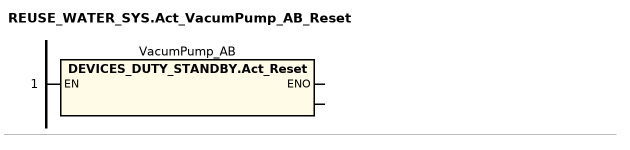
[picture p24: REUSE_WATER_SYS.Act_VacumPump_AB_Reset (LD)]
_LD_ (* Ladder Diagram *)
NETWORK 1
	*
		EN --- VacumPump_AB:DEVICES_DUTY_STANDBY.Act_Reset()
_END_LD_
(* the same logic as Structured Text *)
(* Network 1 *)
VacumPump_AB();
END_ACTION
ACTION Act_VacumPump_AB_Start:
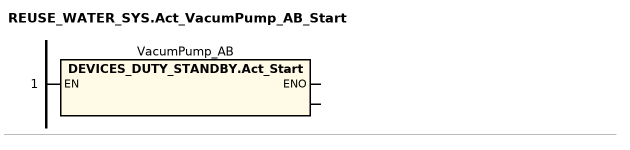
_LD_ (* Ladder Diagram *)
NETWORK 1
	*
		EN --- VacumPump_AB:DEVICES_DUTY_STANDBY.Act_Start()
_END_LD_
(* the same logic as Structured Text *)
(* Network 1 *)
VacumPump_AB();
END_ACTION
ACTION Act_VacumPump_AB_Stop:
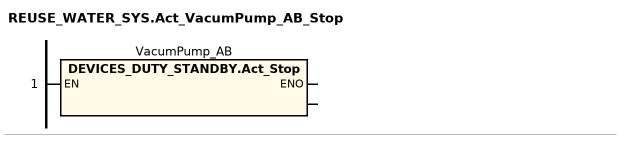
_LD_ (* Ladder Diagram *)
NETWORK 1
	*
		EN --- VacumPump_AB:DEVICES_DUTY_STANDBY.Act_Stop()
_END_LD_
(* the same logic as Structured Text *)
(* Network 1 *)
VacumPump_AB();
END_ACTION
ACTION Control:
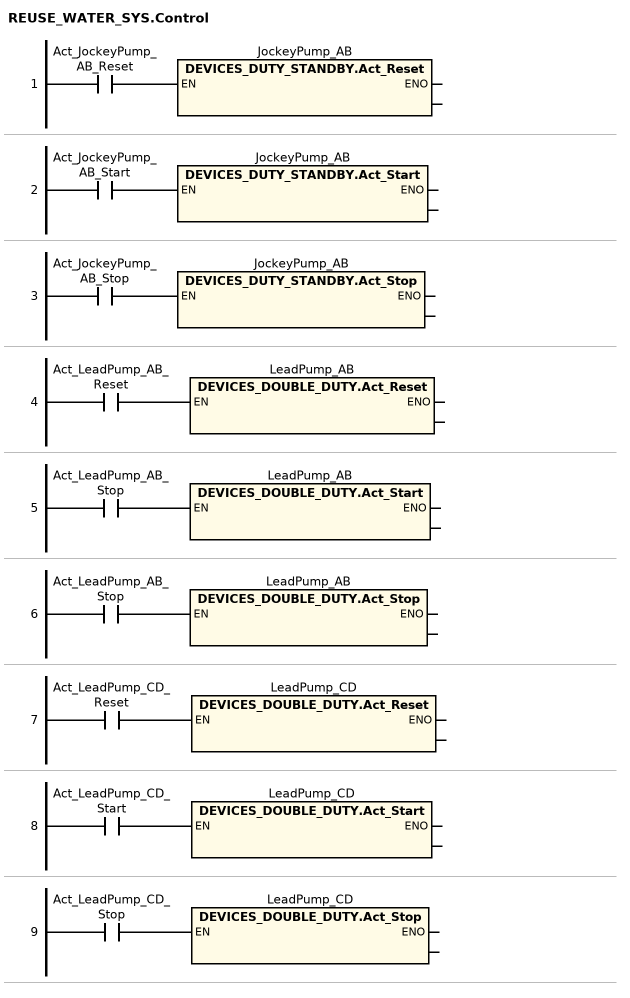
_LD_ (* Ladder Diagram *)
NETWORK 1
	[Act_JockeyPump_AB_Reset]
		EN --- JockeyPump_AB:DEVICES_DUTY_STANDBY.Act_Reset()
NETWORK 2
	[Act_JockeyPump_AB_Start]
		EN --- JockeyPump_AB:DEVICES_DUTY_STANDBY.Act_Start()
NETWORK 3
	[Act_JockeyPump_AB_Stop]
		EN --- JockeyPump_AB:DEVICES_DUTY_STANDBY.Act_Stop()
NETWORK 4
	[Act_LeadPump_AB_Reset]
		EN --- LeadPump_AB:DEVICES_DOUBLE_DUTY.Act_Reset()
NETWORK 5
	[Act_LeadPump_AB_Stop]
		EN --- LeadPump_AB:DEVICES_DOUBLE_DUTY.Act_Start()
NETWORK 6
	[Act_LeadPump_AB_Stop]
		EN --- LeadPump_AB:DEVICES_DOUBLE_DUTY.Act_Stop()
NETWORK 7
	[Act_LeadPump_CD_Reset]
		EN --- LeadPump_CD:DEVICES_DOUBLE_DUTY.Act_Reset()
NETWORK 8
	[Act_LeadPump_CD_Start]
		EN --- LeadPump_CD:DEVICES_DOUBLE_DUTY.Act_Start()
NETWORK 9
	[Act_LeadPump_CD_Stop]
		EN --- LeadPump_CD:DEVICES_DOUBLE_DUTY.Act_Stop()
_END_LD_
(* the same logic as Structured Text *)
(* Network 1 *)
IF Act_JockeyPump_AB_Reset THEN
	JockeyPump_AB();
END_IF;
(* Network 2 *)
IF Act_JockeyPump_AB_Start THEN
	JockeyPump_AB();
END_IF;
(* Network 3 *)
IF Act_JockeyPump_AB_Stop THEN
	JockeyPump_AB();
END_IF;
(* Network 4 *)
IF Act_LeadPump_AB_Reset THEN
	LeadPump_AB();
END_IF;
(* Network 5 *)
IF Act_LeadPump_AB_Stop THEN
	LeadPump_AB();
END_IF;
(* Network 6 *)
IF Act_LeadPump_AB_Stop THEN
	LeadPump_AB();
END_IF;
(* Network 7 *)
IF Act_LeadPump_CD_Reset THEN
	LeadPump_CD();
END_IF;
(* Network 8 *)
IF Act_LeadPump_CD_Start THEN
	LeadPump_CD();
END_IF;
(* Network 9 *)
IF Act_LeadPump_CD_Stop THEN
	LeadPump_CD();
END_IF;
END_ACTION

(* POU SCREENING_OPERATION, SFC *)
FUNCTION_BLOCK SCREENING_OPERATION
VAR_INPUT
END_VAR
VAR_OUTPUT
END_VAR
VAR
	Reset: BOOL;
	PenstockDuty: Penstock;
	PDOpen: BOOL;

	PenstockStandby: Penstock;
	PSOpen: BOOL;

END_VAR
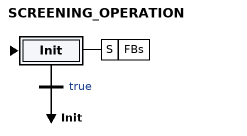
INITIAL_STEP Init:
	FBs(S);
END_STEP
TRANSITION FROM Init TO Init := true;
END_TRANSITION
END_FUNCTION_BLOCK
ACTION FBs:
PenstockDuty(Open:=PDOpen,Reset:=Reset );
PenstockStandby(Open:=PSOpen , Reset:=Reset );
END_ACTION

(* POU Penstock, SFC *)
FUNCTION_BLOCK Penstock
VAR_INPUT
	Open: BOOL;
	Reset: BOOL;
END_VAR
VAR_OUTPUT
END_VAR
VAR
	Warning_PenstockCannotClose:BOOL;
	Warning_PenstockCannotOpen:BOOL;
	Penstock:BOOL;
	PenstockStatus:BOOL;
END_VAR
VAR_IN_OUT
END_VAR
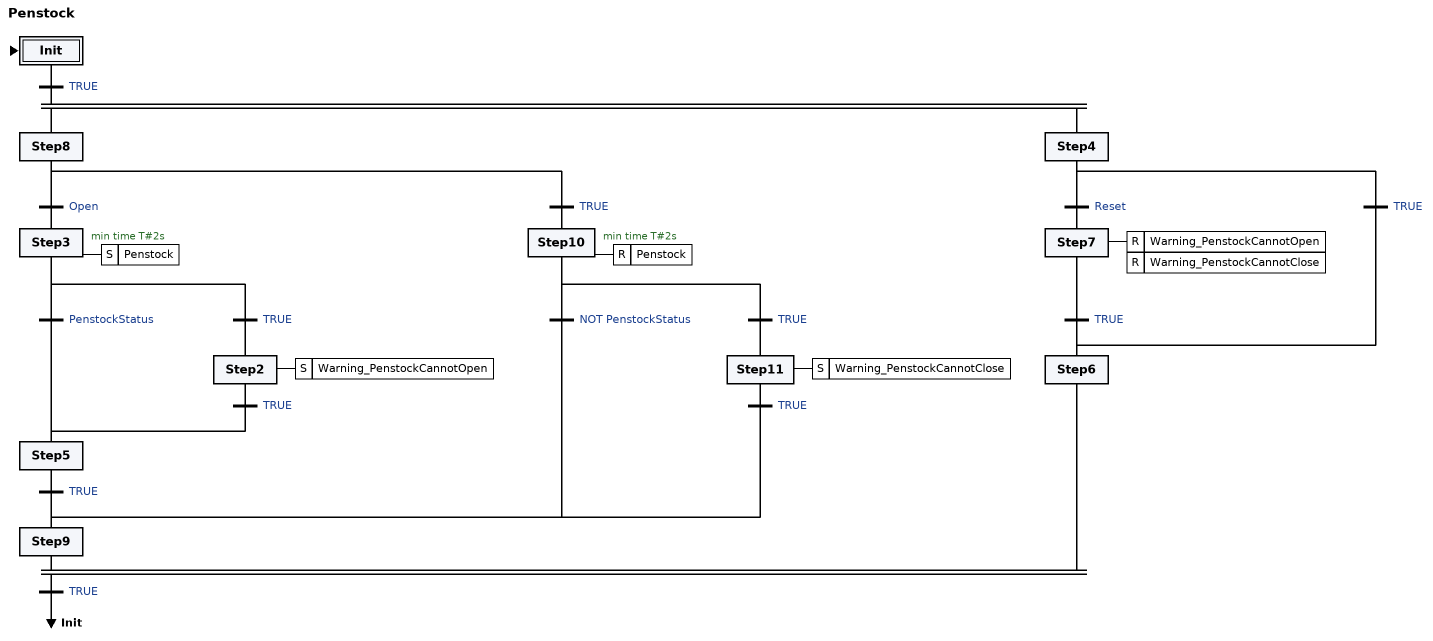
INITIAL_STEP Init:
END_STEP
TRANSITION FROM Init TO (Step8, Step4) := TRUE;
END_TRANSITION
STEP Step8:
END_STEP
TRANSITION FROM Step8 TO Step3 := Open;
END_TRANSITION
TRANSITION FROM Step8 TO Step10 := TRUE;
END_TRANSITION
STEP Step3: (* min time T#2s *)
	Penstock(S);
END_STEP
TRANSITION FROM Step3 TO Step5 := PenstockStatus;
END_TRANSITION
TRANSITION FROM Step3 TO Step2 := TRUE;
END_TRANSITION
STEP Step2:
	Warning_PenstockCannotOpen(S);
END_STEP
TRANSITION FROM Step2 TO Step5 := TRUE;
END_TRANSITION
STEP Step5:
END_STEP
TRANSITION FROM Step5 TO Step9 := TRUE;
END_TRANSITION
STEP Step10: (* min time T#2s *)
	Penstock(R);
END_STEP
TRANSITION FROM Step10 TO Step9 := NOT PenstockStatus;
END_TRANSITION
TRANSITION FROM Step10 TO Step11 := TRUE;
END_TRANSITION
STEP Step11:
	Warning_PenstockCannotClose(S);
END_STEP
TRANSITION FROM Step11 TO Step9 := TRUE;
END_TRANSITION
STEP Step9:
END_STEP
STEP Step4:
END_STEP
TRANSITION FROM Step4 TO Step7 := Reset;
END_TRANSITION
TRANSITION FROM Step4 TO Step6 := TRUE;
END_TRANSITION
STEP Step7:
	Warning_PenstockCannotOpen(R);
	Warning_PenstockCannotClose(R);
END_STEP
TRANSITION FROM Step7 TO Step6 := TRUE;
END_TRANSITION
STEP Step6:
END_STEP
TRANSITION FROM (Step9, Step6) TO Init := TRUE;
END_TRANSITION
END_FUNCTION_BLOCK

(* POU DEVICES_FINE_SCREEN, SFC *)
FUNCTION_BLOCK DEVICES_FINE_SCREEN
VAR

	Duty_RemoteMode AT%I*: BOOL;
	Duty_CommandStart AT%I*: BOOL;
	Duty_Overload AT%I*: BOOL;
	Duty_Incomplete AT%I*: BOOL;
	Duty_StartStatus AT%I*: BOOL;


	Done_StartStandby: BOOL;
	Done_Start: BOOL;
	Done_Stop: BOOL;


	Duty2_CommandStart AT%I*: BOOL;
	Duty2_RemoteMode AT%I*: BOOL;
	Duty2_Overload AT%I*: BOOL;
	Duty2_Incomplete AT%I*: BOOL;
	Duty2_StartStatus AT%I*: BOOL;

	Warning_DutyFailed: BOOL;
	Warning_Duty2Failed: BOOL;
	CriticalAlarm_Duty2CannotStop : BOOL;
	CriticalAlarm_DutyCannotStop : BOOL;

END_VAR
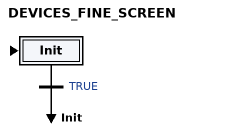
INITIAL_STEP Init:
END_STEP
TRANSITION FROM Init TO Init := TRUE;
END_TRANSITION
END_FUNCTION_BLOCK
ACTION Act_Reset:
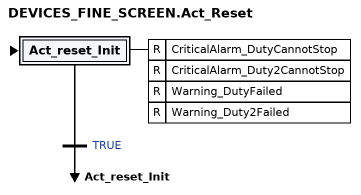
INITIAL_STEP Act_reset_Init:
	CriticalAlarm_DutyCannotStop(R);
	CriticalAlarm_Duty2CannotStop(R);
	Warning_DutyFailed(R);
	Warning_Duty2Failed(R);
END_STEP
TRANSITION FROM Act_reset_Init TO Act_reset_Init := TRUE;
END_TRANSITION
END_ACTION
ACTION Act_Start:
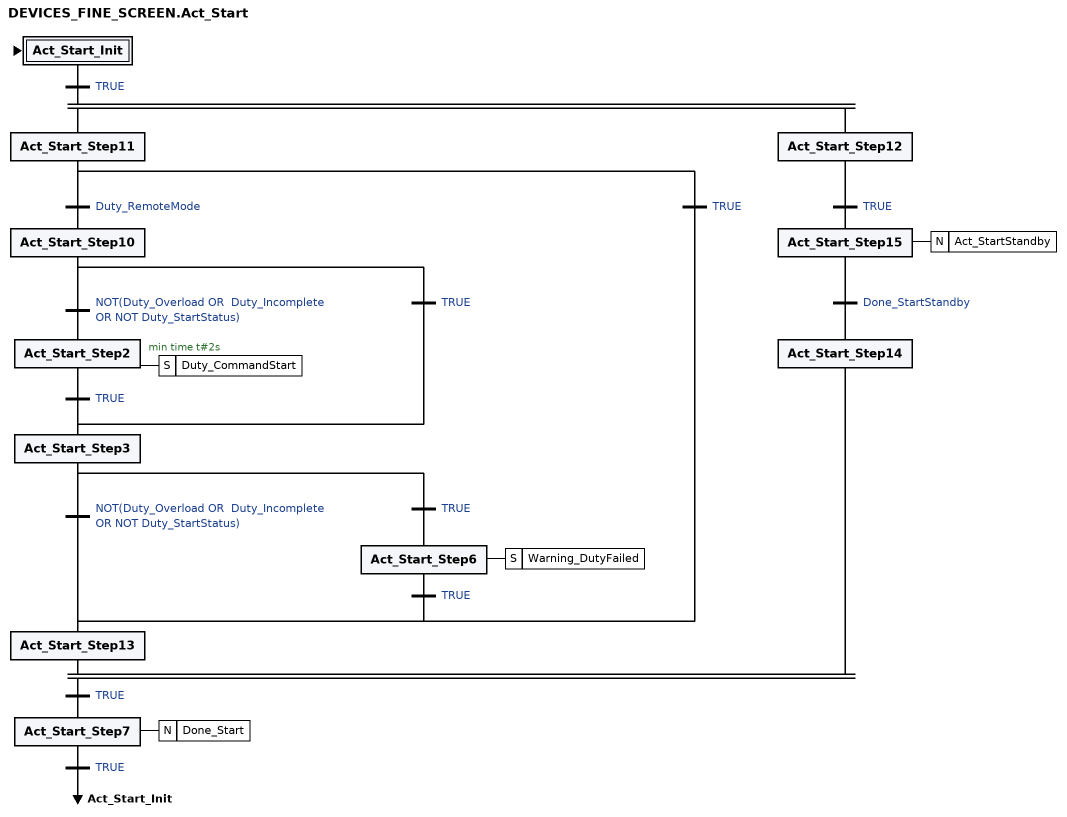
INITIAL_STEP Act_Start_Init:
END_STEP
TRANSITION FROM Act_Start_Init TO (Act_Start_Step11, Act_Start_Step12) := TRUE;
END_TRANSITION
STEP Act_Start_Step11:
END_STEP
TRANSITION FROM Act_Start_Step11 TO Act_Start_Step10 := Duty_RemoteMode;
END_TRANSITION
TRANSITION FROM Act_Start_Step11 TO Act_Start_Step13 := TRUE;
END_TRANSITION
STEP Act_Start_Step10:
END_STEP
TRANSITION FROM Act_Start_Step10 TO Act_Start_Step2 := NOT(Duty_Overload OR  Duty_Incomplete OR NOT Duty_StartStatus);
END_TRANSITION
TRANSITION FROM Act_Start_Step10 TO Act_Start_Step3 := TRUE;
END_TRANSITION
STEP Act_Start_Step2: (* min time t#2s *)
	Duty_CommandStart(S);
END_STEP
TRANSITION FROM Act_Start_Step2 TO Act_Start_Step3 := TRUE;
END_TRANSITION
STEP Act_Start_Step3:
END_STEP
TRANSITION FROM Act_Start_Step3 TO Act_Start_Step13 := NOT(Duty_Overload OR  Duty_Incomplete OR NOT Duty_StartStatus);
END_TRANSITION
TRANSITION FROM Act_Start_Step3 TO Act_Start_Step6 := TRUE;
END_TRANSITION
STEP Act_Start_Step6:
	Warning_DutyFailed(S);
END_STEP
TRANSITION FROM Act_Start_Step6 TO Act_Start_Step13 := TRUE;
END_TRANSITION
STEP Act_Start_Step13:
END_STEP
STEP Act_Start_Step12:
END_STEP
TRANSITION FROM Act_Start_Step12 TO Act_Start_Step15 := TRUE;
END_TRANSITION
STEP Act_Start_Step15:
	Act_StartStandby(N);
END_STEP
TRANSITION FROM Act_Start_Step15 TO Act_Start_Step14 := Done_StartStandby;
END_TRANSITION
STEP Act_Start_Step14:
END_STEP
TRANSITION FROM (Act_Start_Step13, Act_Start_Step14) TO Act_Start_Step7 := TRUE;
END_TRANSITION
STEP Act_Start_Step7:
	Done_Start(N);
END_STEP
TRANSITION FROM Act_Start_Step7 TO Act_Start_Init := TRUE;
END_TRANSITION
END_ACTION
ACTION Act_StartStandby:
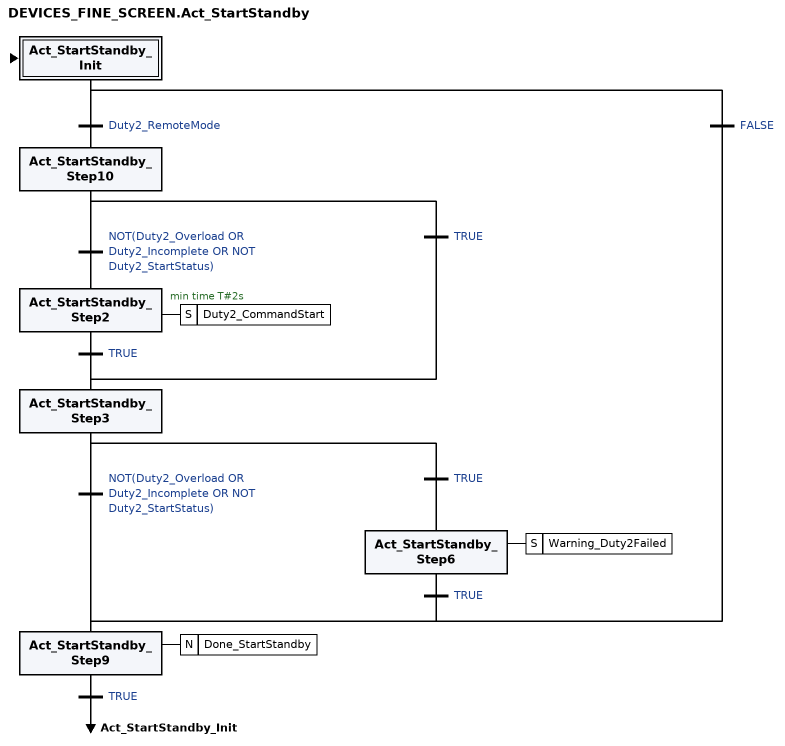
INITIAL_STEP Act_StartStandby_Init:
END_STEP
TRANSITION FROM Act_StartStandby_Init TO Act_StartStandby_Step10 := Duty2_RemoteMode;
END_TRANSITION
TRANSITION FROM Act_StartStandby_Init TO Act_StartStandby_Step9 := FALSE;
END_TRANSITION
STEP Act_StartStandby_Step10:
END_STEP
TRANSITION FROM Act_StartStandby_Step10 TO Act_StartStandby_Step2 := NOT(Duty2_Overload OR  Duty2_Incomplete OR NOT Duty2_StartStatus);
END_TRANSITION
TRANSITION FROM Act_StartStandby_Step10 TO Act_StartStandby_Step3 := TRUE;
END_TRANSITION
STEP Act_StartStandby_Step2: (* min time T#2s *)
	Duty2_CommandStart(S);
END_STEP
TRANSITION FROM Act_StartStandby_Step2 TO Act_StartStandby_Step3 := TRUE;
END_TRANSITION
STEP Act_StartStandby_Step3:
END_STEP
TRANSITION FROM Act_StartStandby_Step3 TO Act_StartStandby_Step9 := NOT(Duty2_Overload OR  Duty2_Incomplete OR NOT Duty2_StartStatus);
END_TRANSITION
TRANSITION FROM Act_StartStandby_Step3 TO Act_StartStandby_Step6 := TRUE;
END_TRANSITION
STEP Act_StartStandby_Step6:
	Warning_Duty2Failed(S);
END_STEP
TRANSITION FROM Act_StartStandby_Step6 TO Act_StartStandby_Step9 := TRUE;
END_TRANSITION
STEP Act_StartStandby_Step9:
	Done_StartStandby(N);
END_STEP
TRANSITION FROM Act_StartStandby_Step9 TO Act_StartStandby_Init := TRUE;
END_TRANSITION
END_ACTION
ACTION Act_Stop:
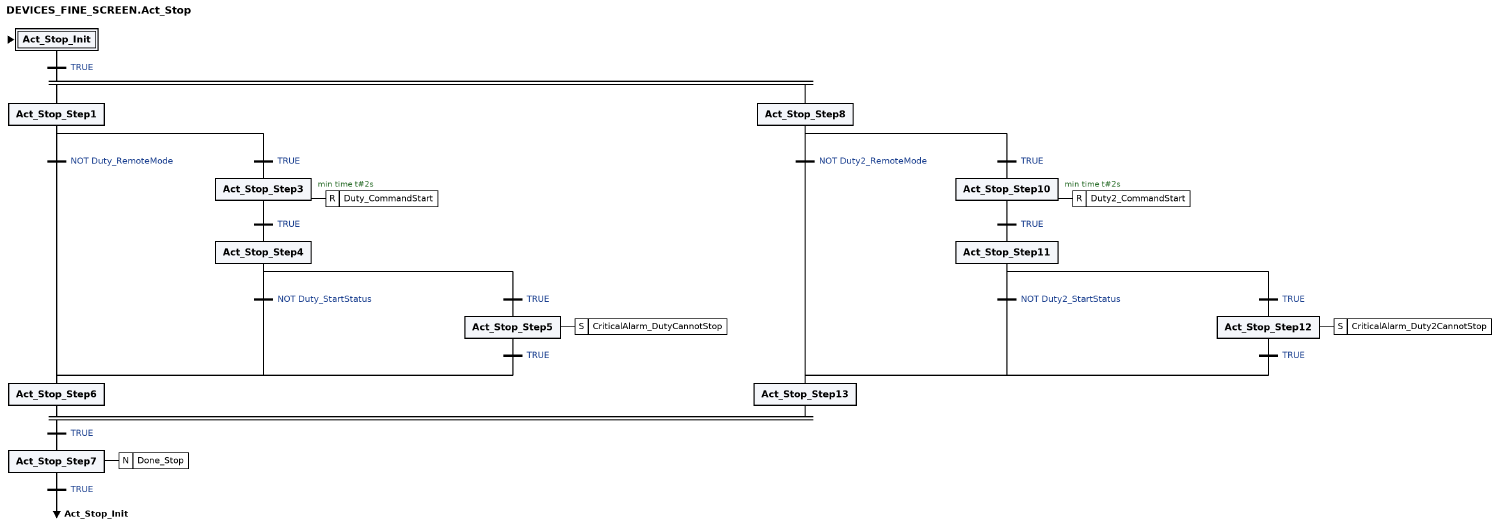
INITIAL_STEP Act_Stop_Init:
END_STEP
TRANSITION FROM Act_Stop_Init TO (Act_Stop_Step1, Act_Stop_Step8) := TRUE;
END_TRANSITION
STEP Act_Stop_Step1:
END_STEP
TRANSITION FROM Act_Stop_Step1 TO Act_Stop_Step6 := NOT Duty_RemoteMode;
END_TRANSITION
TRANSITION FROM Act_Stop_Step1 TO Act_Stop_Step3 := TRUE;
END_TRANSITION
STEP Act_Stop_Step3: (* min time t#2s *)
	Duty_CommandStart(R);
END_STEP
TRANSITION FROM Act_Stop_Step3 TO Act_Stop_Step4 := TRUE;
END_TRANSITION
STEP Act_Stop_Step4:
END_STEP
TRANSITION FROM Act_Stop_Step4 TO Act_Stop_Step6 := NOT Duty_StartStatus;
END_TRANSITION
TRANSITION FROM Act_Stop_Step4 TO Act_Stop_Step5 := TRUE;
END_TRANSITION
STEP Act_Stop_Step5:
	CriticalAlarm_DutyCannotStop(S);
END_STEP
TRANSITION FROM Act_Stop_Step5 TO Act_Stop_Step6 := TRUE;
END_TRANSITION
STEP Act_Stop_Step6:
END_STEP
STEP Act_Stop_Step8:
END_STEP
TRANSITION FROM Act_Stop_Step8 TO Act_Stop_Step13 := NOT Duty2_RemoteMode;
END_TRANSITION
TRANSITION FROM Act_Stop_Step8 TO Act_Stop_Step10 := TRUE;
END_TRANSITION
STEP Act_Stop_Step10: (* min time t#2s *)
	Duty2_CommandStart(R);
END_STEP
TRANSITION FROM Act_Stop_Step10 TO Act_Stop_Step11 := TRUE;
END_TRANSITION
STEP Act_Stop_Step11:
END_STEP
TRANSITION FROM Act_Stop_Step11 TO Act_Stop_Step13 := NOT Duty2_StartStatus;
END_TRANSITION
TRANSITION FROM Act_Stop_Step11 TO Act_Stop_Step12 := TRUE;
END_TRANSITION
STEP Act_Stop_Step12:
	CriticalAlarm_Duty2CannotStop(S);
END_STEP
TRANSITION FROM Act_Stop_Step12 TO Act_Stop_Step13 := TRUE;
END_TRANSITION
STEP Act_Stop_Step13:
END_STEP
TRANSITION FROM (Act_Stop_Step6, Act_Stop_Step13) TO Act_Stop_Step7 := TRUE;
END_TRANSITION
STEP Act_Stop_Step7:
	Done_Stop(N);
END_STEP
TRANSITION FROM Act_Stop_Step7 TO Act_Stop_Init := TRUE;
END_TRANSITION
END_ACTION
